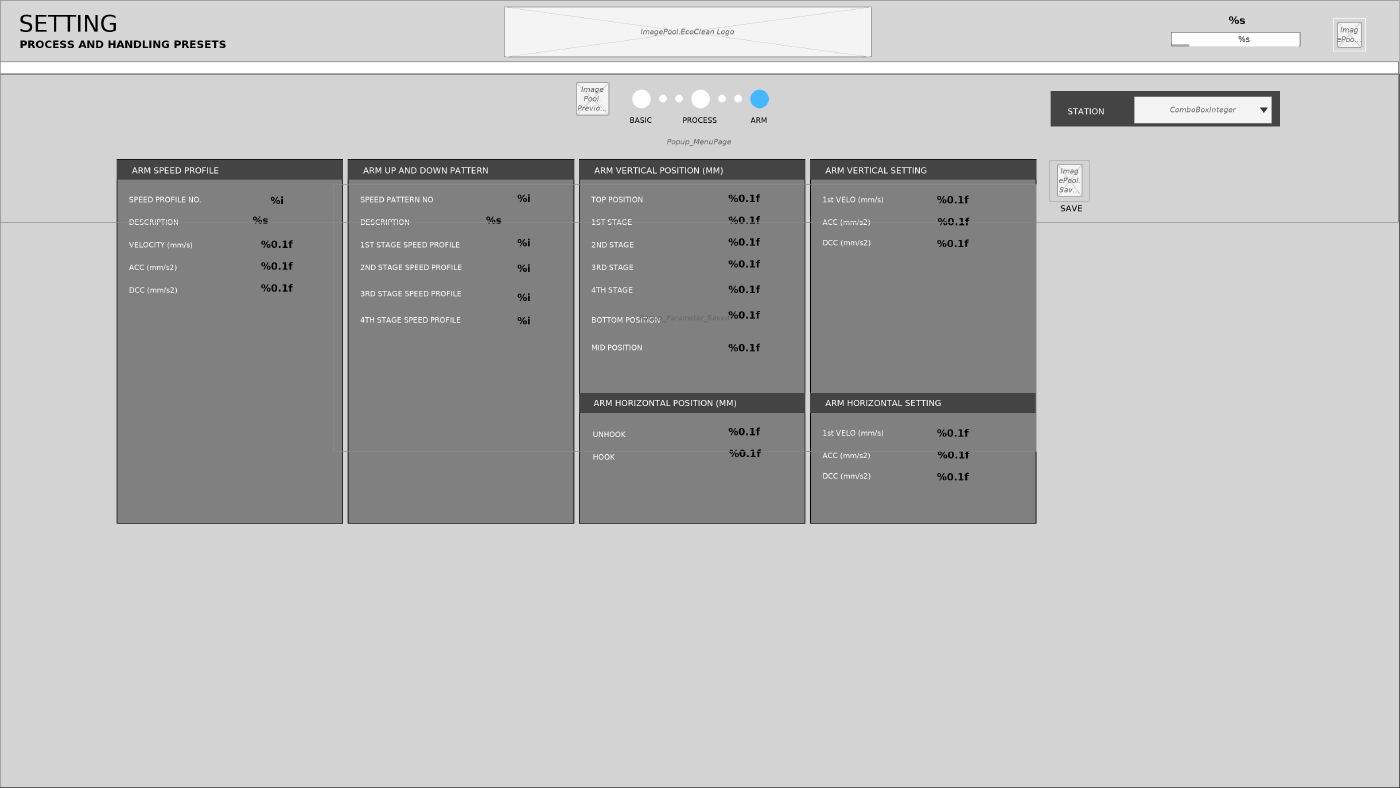
VISUALIZATION SettingArm_Page  // 1920x1081
    Rectangle (0,101 1920x980)
    Rectangle (0,63 1920x26)
        p3528305787: HMI_Ctrl.ANIMATION3
    Rectangle (0,0 1919x85)
    Label (23,6 267x53), "SETTING"
    Label (24,49 320x24), "PROCESS AND HANDLING PRESETS"
    Group (1828,25 45x45)
        OnMouseClick: toggle HMI_Ctrl.MenuButton
        RoundedRectangle (0,0 45x45), colour toggle: HMI_Ctrl.MenuButton
        Image (6,5 33x35), image: ImagePool.Menu Button
    Ellipse (867,123 25x25)
    Ellipse (948,123 25x25)
    Ellipse (904,130 10x10)
    Ellipse (926,130 10x10)
    Ellipse (985,130 10x10)
    Ellipse (1007,130 10x10)
    Ellipse (1029,123 25x25)
    Label (847,153 64x24), "BASIC"
    Label (928,153 64x24), "PROCESS"
    Label (1009,153 64x24), "ARM"
    Image (790,113 45x45), image: ImagePool.Previous Button
        OnMouseClick: change screen: SettingProcess_Page
    RoundedRectangle (1441,125 314x48)
    ComboBoxInteger (1555,132 189x37), variable: iArmSettingStnNoBuffer, text list: 'TextList_Arm_Setting'
    Label (1461,141 79x24), "STATION"
    Rectangle (160,218 310x500)
    Rectangle (160,219 310x27)
    Label (178,222 143x24), "ARM SPEED PROFILE"
    Label (174,262 141x24), "SPEED PROFILE NO."
    Label (174,293 108x24), "DESCRIPTION"
    Label (174,324 116x24), "VELOCITY (mm/s)"
    Label (174,355 118x24), "ACC (mm/s2)"
    Label (174,386 82x24), "DCC (mm/s2)"
    Rectangle (477,218 310x500)
    Rectangle (477,219 310x27)
    Label (495,222 213x24), "ARM UP AND DOWN PATTERN"
    Rectangle (794,218 310x500)
    Rectangle (794,219 310x27)
    Label (812,222 228x24), "ARM VERTICAL POSITION (MM)"
    Rectangle (1111,218 310x500)
    Rectangle (1111,219 310x27)
    Label (1129,222 200x24), "ARM VERTICAL SETTING"
    Label (1125,262 109x24), "1st VELO (mm/s)"
    Label (1125,293 108x24), "ACC (mm/s2)"
    Label (491,262 147x24), "SPEED PATTERN NO"
    Label (491,293 108x24), "DESCRIPTION"
    Label (491,324 196x24), "1ST STAGE SPEED PROFILE"
    Label (491,355 186x24), "2ND STAGE SPEED PROFILE"
    Label (491,391 186x24), "3RD STAGE SPEED PROFILE"
    Label (491,427 186x24), "4TH STAGE SPEED PROFILE"
    Label (808,262 147x24), "TOP POSITION"
    Label (808,293 108x24), "1ST STAGE"
    Label (808,324 196x24), "2ND STAGE"
    Label (808,355 186x24), "3RD STAGE"
    Label (808,386 186x24), "4TH STAGE"
    Label (808,427 186x24), "BOTTOM POSITION"
    Rectangle (1111,539 310x27)
    Label (1129,541 200x24), "ARM HORIZONTAL SETTING"
    Rectangle (310,267 140x17), "%i", text variable: DSA31ArmSpeedProfileStore.iArmSpdProfileNo, input disabled if: bMainOnOff
        OnMouseDown: write the text variable via VisuDialogs.Numpad, min 1, max 20
    Rectangle (263,294 189x17), "%s", text variable: DSA31ArmSpeedProfileStore.DsArmSpeedProfile.sDescription, input disabled if: bMainOnOff
        OnMouseDown: write the text variable via VisuDialogs.Keypad
    Rectangle (310,327 140x17), "%0.1f", text variable: DSA31ArmSpeedProfileStore.DsArmSpeedProfile.lrSpeedVelo, input disabled if: bMainOnOff
        OnMouseDown: write the text variable via VisuDialogs.Numpad, min 2, max 400
    Rectangle (310,357 140x17), "%0.1f", text variable: DSA31ArmSpeedProfileStore.DsArmSpeedProfile.lrAcc, input disabled if: bMainOnOff
        OnMouseDown: write the text variable via VisuDialogs.Numpad, min 100, max 1500
    Rectangle (310,387 140x17), "%0.1f", text variable: DSA31ArmSpeedProfileStore.DsArmSpeedProfile.lrDcc, input disabled if: bMainOnOff
        OnMouseDown: write the text variable via VisuDialogs.Numpad, min 100, max 1500
    Rectangle (653,264 131x17), "%i", text variable: DSA21UpDownPatternStore.iUpDownPatternNo, input disabled if: bMainOnOff
        OnMouseDown: write the text variable via VisuDialogs.Numpad, min 1, max 20
    Rectangle (654,325 129x17), "%i", text variable: DSA21UpDownPatternStore.DsInUpDownPatternMemory.iZone1SpdProfileNo, input disabled if: bMainOnOff
        OnMouseDown: write the text variable via VisuDialogs.Numpad, min 1, max 20
    Rectangle (654,360 129x17), "%i", text variable: DSA21UpDownPatternStore.DsInUpDownPatternMemory.iZone2SpdProfileNo, input disabled if: bMainOnOff
        OnMouseDown: write the text variable via VisuDialogs.Numpad, min 1, max 20
    Rectangle (654,400 129x17), "%i", text variable: DSA21UpDownPatternStore.DsInUpDownPatternMemory.iZone3SpdProfileNo, input disabled if: bMainOnOff
        OnMouseDown: write the text variable via VisuDialogs.Numpad, min 1, max 20
    Rectangle (654,432 129x17), "%i", text variable: DSA21UpDownPatternStore.DsInUpDownPatternMemory.iZone4SpdProfileNo, input disabled if: bMainOnOff
        OnMouseDown: write the text variable via VisuDialogs.Numpad, min 1, max 20
    Rectangle (583,294 189x17), "%s", text variable: DSA21UpDownPatternStore.DsInUpDownPatternMemory.sDescription, input disabled if: bMainOnOff
        OnMouseDown: write the text variable via VisuDialogs.Keypad
    Rectangle (951,264 140x17), "%0.1f", text variable: Arm1TopPos[iArmSettingStnNo], input disabled if: bMainOnOff
        OnMouseDown: write the text variable via VisuDialogs.Numpad
    Rectangle (951,294 140x17), "%0.1f", text variable: Arm1Pos1stStage[iArmSettingStnNo], input disabled if: bMainOnOff
        OnMouseDown: write the text variable via VisuDialogs.Numpad
    Rectangle (951,324 140x17), "%0.1f", text variable: Arm1Pos2ndStage[iArmSettingStnNo], input disabled if: bMainOnOff
        OnMouseDown: write the text variable via VisuDialogs.Numpad
    Rectangle (951,354 140x17), "%0.1f", text variable: Arm1Pos3rdStage[iArmSettingStnNo], input disabled if: bMainOnOff
        OnMouseDown: write the text variable via VisuDialogs.Numpad
    Rectangle (951,389 140x17), "%0.1f", text variable: Arm1Pos4thStage[iArmSettingStnNo], input disabled if: bMainOnOff
        OnMouseDown: write the text variable via VisuDialogs.Numpad
    Rectangle (951,424 140x17), "%0.1f", text variable: Arm1BottomPos[iArmSettingStnNo], input disabled if: bMainOnOff
        OnMouseDown: write the text variable via VisuDialogs.Numpad
    Rectangle (794,539 310x27)
    Label (811,541 228x24), "ARM HORIZONTAL POSITION (MM)"
    Label (810,584 109x24), "UNHOOK"
    Label (810,615 108x24), "HOOK"
    Rectangle (951,584 140x17), "%0.1f", text variable: Arm1UnHookPos[iArmSettingStnNo], input disabled if: bMainOnOff
        OnMouseDown: write the text variable via VisuDialogs.Numpad
    Rectangle (952,614 140x17), "%0.1f", text variable: Arm1HookPos[iArmSettingStnNo], input disabled if: bMainOnOff
        OnMouseDown: write the text variable via VisuDialogs.Numpad
    Label (1125,321 108x24), "DCC (mm/s2)"
    Rectangle (1237,266 140x17), "%0.1f", text variable: ARlrVertPos_In_HighSpeed[1], input disabled if: bMainOnOff
        OnMouseDown: write the text variable via VisuDialogs.Numpad, min 2, max 400
    Rectangle (1238,296 140x17), "%0.1f", text variable: ARlrVertPos_In_Acc[1], input disabled if: bMainOnOff
        OnMouseDown: write the text variable via VisuDialogs.Numpad, min 200, max 1500
    Rectangle (1237,326 140x17), "%0.1f", text variable: ARlrVertPos_In_Dcc[1], input disabled if: bMainOnOff
        OnMouseDown: write the text variable via VisuDialogs.Numpad, min 200, max 1500
    Label (1125,582 109x24), "1st VELO (mm/s)"
    Label (1125,613 108x24), "ACC (mm/s2)"
    Label (1125,641 108x24), "DCC (mm/s2)"
    Rectangle (1237,586 140x17), "%0.1f", text variable: ARlrHorzPos_In_HighSpeed[1], input disabled if: bMainOnOff
        OnMouseDown: write the text variable via VisuDialogs.Numpad, min 50, max 600
    Rectangle (1238,616 140x17), "%0.1f", text variable: ARlrHorzPos_In_Acc[1], input disabled if: bMainOnOff
        OnMouseDown: write the text variable via VisuDialogs.Numpad, min 200, max 1500
    Rectangle (1237,646 140x17), "%0.1f", text variable: ARlrHorzPos_In_Dcc[1], input disabled if: bMainOnOff
        OnMouseDown: write the text variable via VisuDialogs.Numpad, min 200, max 1500
    Image (691,9 504x69), image: ImagePool.EcoClean Logo
    Label (808,465 186x24), "MID POSITION", invisible if: iArmSettingStnNo<>9
    Rectangle (951,469 140x17), "%0.1f", text variable: Arm1MidPos[iArmSettingStnNo], invisible if: iArmSettingStnNo<>9, input disabled if: bMainOnOff
        OnMouseDown: write the text variable via VisuDialogs.Numpad
    Group (1606,17 179x46)
        Button (0,27 177x19), image: VisuSymbols.Symbols.AddUser
        Rectangle (25,28 150x18), "%s", text variable: fbHmiTF1800_UserlevelManagement.dsHmiUserStatus_Active.sLoginName
        Rectangle (2,0 177x22), "%s", text variable: DSLocalSystemTimeML.sCurrentDT24Hr_General
    Group (1439,220 56x80), invisible if: bMainOnOff
        Label (5,52 51x28), "SAVE", invisible if: bMainOnOff
        RoundedRectangle (0,0 55x56), colour toggle: bRecipeSavePb
            tap bRecipeSavePb
        Image (11,5 34x45), image: ImagePool.Save Button
            OnMouseDown: execute { bRecipeSavePb:=1; }
            OnMouseUp: execute { bRecipeSavePb:=0; }
    Frame (457,253 964x366), invisible if: NOT stWritePersistentData.SaveHR
        shows Popup_Parameter_Saved()
    Frame (0,84 1918x221), invisible if: HMI_Ctrl.CloseMenuButton
        shows Popup_MenuPage()
END_VISUALIZATION

(* stored: Version 1.1.0.1, ProductVersion 3.1.4024.12
   Visu SettingArm_Page: Id {397abe47-e8c0-4595-989b-cc3fb73e3772} *)
